FUNCTION_BLOCK DataTypesTime (* Template for an empty basic function block *)
  (* Standard: 61499-2; Description: Copyright (c) 2019 Jan Holzweber This program and the accompanying materials are made available under the terms of the Eclipse Public License 2.0 which is available at https://www.eclipse.org/legal/epl-2.0/ SPDX-License-Identifier: EPL-2.0 *)
  (* Version 1.0, 2019-06-05, jholz *)
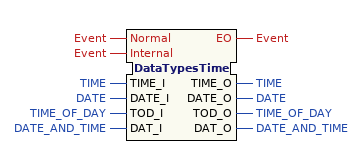
  EVENT_INPUT
    Normal;
    Internal;
  END_EVENT
  EVENT_OUTPUT
    EO;
  END_EVENT
  VAR_INPUT
    TIME_I : TIME;
    DATE_I : DATE;
    TOD_I : TIME_OF_DAY;
    DAT_I : DATE_AND_TIME;
  END_VAR
  VAR_OUTPUT
    TIME_O : TIME;
    DATE_O : DATE;
    TOD_O : TIME_OF_DAY;
    DAT_O : DATE_AND_TIME;
  END_VAR
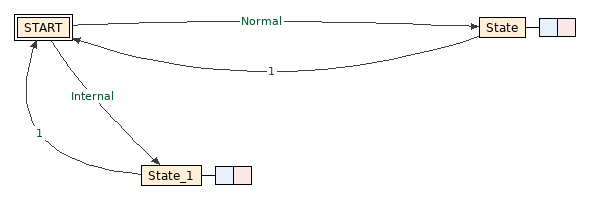
  EC_STATES
    START; (* Initial State *)
    State;
    State_1;
  END_STATES
  EC_TRANSITIONS
    START TO State := Normal;
    State TO START := 1;
    START TO State_1 := Internal;
    State_1 TO START := 1;
  END_TRANSITIONS
  ALGORITHM Normal IN ST: (* new algorithm *)
TIME_O:=TIME_I;
DATE_O:=DATE_I;
TOD_O:=TOD_I;
DAT_O:=DAT_I;
  END_ALGORITHM
  ALGORITHM Internal IN ST: (* new algorithm *)
TIME_O:=TIME#1m;
DATE_O:=D#1996-08-12;
TOD_O:=TOD#06:06:66;
DAT_O:=DT#1989-06-15-13:56:14.77;
  END_ALGORITHM
END_FUNCTION_BLOCK
